FUNCTION_BLOCK FB_MotionClearAsserts_Test EXTENDS TcUnit.FB_TestSuite
VAR
END_VAR


TestBasic();

METHOD TestBasic
VAR
    nIter: UINT;
END_VAR
VAR_INST
    fbClear: FB_MotionClearAsserts;
    astDbStateParams: ARRAY[0..GeneralConstants.MAX_STATES] OF ST_DbStateParams;
    fbArbiter: FB_Arbiter(1);
END_VAR

TEST('TestBasic');

FOR nIter := 0 TO GeneralConstants.MAX_STATES DO
    astDbStateParams[nIter].nRequestAssertionID := 100 + nIter;
    fbArbiter.AddRequest(
        nReqID:=100 + nIter,
        stReqBP:=PMPS_GVL.cstFullBeam,
        sDevName:='UnitTest',
    );
END_FOR

FOR nIter := 0 TO GeneralConstants.MAX_STATES DO
    AssertTrue(
        fbArbiter.CheckRequestInPool(100 + nIter),
        CONCAT(CONCAT('State ', UDINT_TO_STRING(nIter)), ' was not in the pool'),
    );
END_FOR

fbClear(
    astDbStateParams:=astDbStateParams,
    fbArbiter:=fbArbiter,
    bExecute:=TRUE,
);

FOR nIter := 0 TO GeneralConstants.MAX_STATES DO
    AssertFalse(
        fbArbiter.CheckRequestInPool(100 + nIter),
        CONCAT(CONCAT('State ', UDINT_TO_STRING(nIter)), ' was not cleared from the pool'),
    );
END_FOR

TEST_FINISHED();
END_METHOD

END_FUNCTION_BLOCK

(* stored: Version 1.1.0.1
   POU FB_MotionClearAsserts_Test: Id {f92faa2f-544b-4cb5-9f0d-b3d1a8e6ba98}, SpecialFunc None
   Method TestBasic: Id {2219d5cb-d17f-45f4-9105-eb6686b76151} *)
